FUNCTION_BLOCK Flash
VAR
	ton1: TON;
	ton2: TON;
END_VAR
VAR_INPUT
	bstart: BOOL;
	Time_off: TIME;
	Time_on: TIME;
END_VAR
VAR_OUTPUT
	out: BOOL;
END_VAR

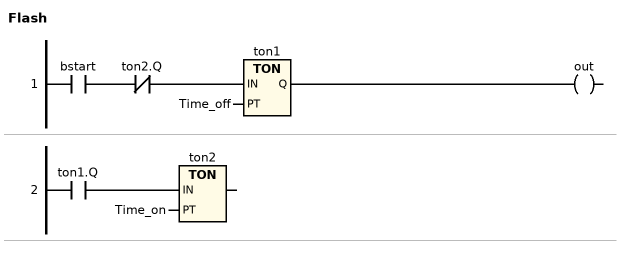
// NETWORK 1
ton1(IN := bstart AND NOT ton2.Q, PT := Time_off); // TON
out := ton1.Q;

// NETWORK 2
ton2(IN := ton1.Q, PT := Time_on); // TON

END_FUNCTION_BLOCK

(* stored: Version 1.1.0.1
   POU Flash: Id {863ef1e9-ff62-412a-a9e7-636748db6f12}, SpecialFunc None *)
